// Mitsubishi GX Works2 project: 3. teaching   PLC: Q03UDV

PROGRAM MAIN
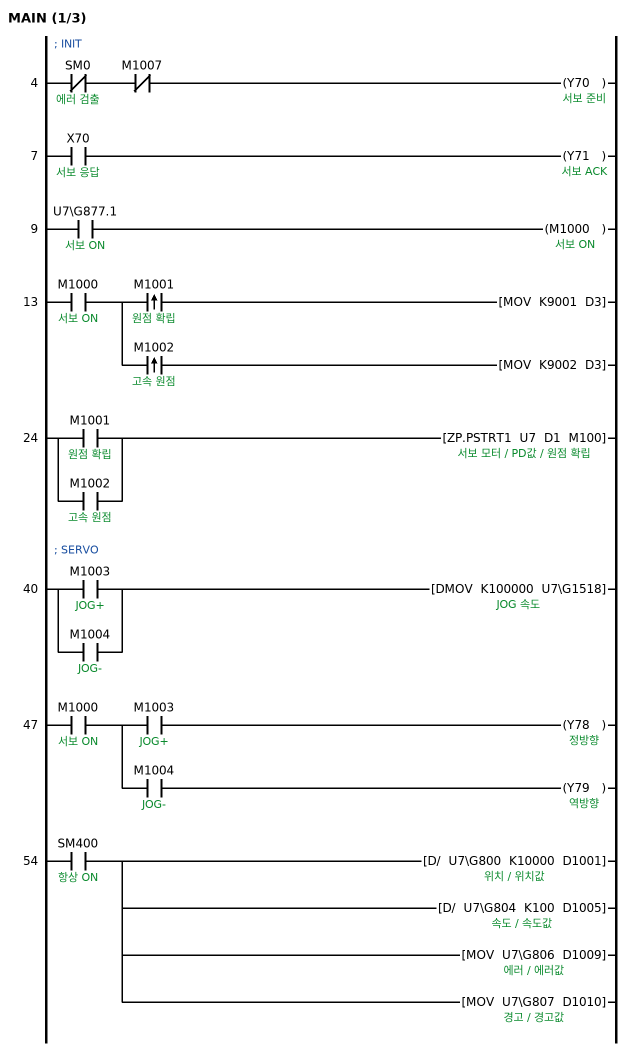
; INIT
4     LDI     SM0  ; 에러 검출
      ANI     M1007
      OUT     Y70  ; 서보 준비
7     LD      X70  ; 서보 응답
      OUT     Y71  ; 서보 ACK
9     LD      U7\G877.1  ; 서보 ON
      OUT     M1000  ; 서보 ON
13    LD      M1000  ; 서보 ON
      MPS
      ANDP    M1001  ; 원점 확립
      MOV     K9001 D3
      MPP
      ANDP    M1002  ; 고속 원점
      MOV     K9002 D3
24    LD      M1001  ; 원점 확립
      OR      M1002  ; 고속 원점
      ZP.PSTRT1 U7 D1 M100  ; 서보 모터 / PD값 / 원점 확립
; SERVO
40    LD      M1003  ; JOG+
      OR      M1004  ; JOG-
      DMOV    K100000 U7\G1518  ; JOG 속도
47    LD      M1000  ; 서보 ON
      MPS
      AND     M1003  ; JOG+
      OUT     Y78  ; 정방향
      MPP
      AND     M1004  ; JOG-
      OUT     Y79  ; 역방향
54    LD      SM400  ; 항상 ON
      D/      U7\G800 K10000 D1001  ; 위치 / 위치값
      D/      U7\G804 K100 D1005  ; 속도 / 속도값
      MOV     U7\G806 D1009  ; 에러 / 에러값
      MOV     U7\G807 D1010  ; 경고 / 경고값
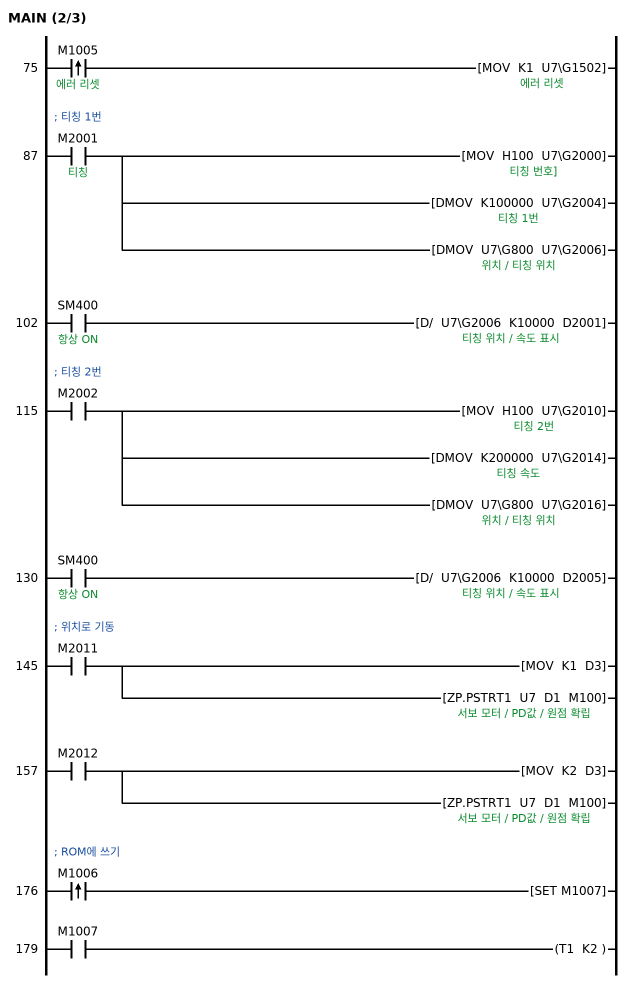
75    LDP     M1005  ; 에러 리셋
      MOV     K1 U7\G1502  ; 에러 리셋
; 티칭 1번
87    LD      M2001  ; 티칭
      MOV     H100 U7\G2000  ; 티칭 번호]
      DMOV    K100000 U7\G2004  ; 티칭 1번
      DMOV    U7\G800 U7\G2006  ; 티칭 위치
102   LD      SM400  ; 항상 ON
      D/      U7\G2006 K10000 D2001  ; 속도 표시
; 티칭 2번
115   LD      M2002
      MOV     H100 U7\G2010  ; 티칭 2번
      DMOV    K200000 U7\G2014  ; 티칭 속도
      DMOV    U7\G800 U7\G2016  ; 티칭 위치
130   LD      SM400  ; 항상 ON
      D/      U7\G2006 K10000 D2005  ; 속도 표시
; 위치로 기동
145   LD      M2011
      MOV     K1 D3
      ZP.PSTRT1 U7 D1 M100
157   LD      M2012
      MOV     K2 D3
      ZP.PSTRT1 U7 D1 M100
; ROM에 쓰기
176   LDP     M1006
      SET     M1007
179   LD      M1007
      OUT     T1 K2
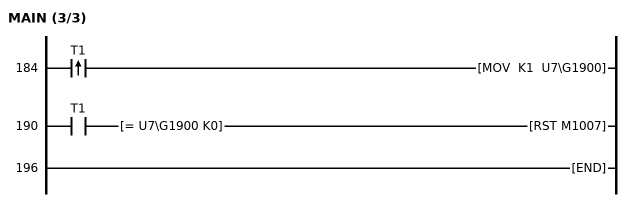
184   LDP     T1
      MOV     K1 U7\G1900
190   LD      T1
      AND=    U7\G1900 K0
      RST     M1007
196   END
END_PROGRAM

// device comments not shown above
X0  ; 공급 후진
X1  ; 공급 전진
X2  ; 분배 후진
X3  ; 분배 전진
X4  ; 가공 상승
X15  ; PB1
X16  ; PB2
X17  ; PB3
X1C  ; Toggle
Y20  ; 공급+
Y21  ; 공급-
Y22  ; 분배+
Y23  ; 분배-
M1  ; 공급+
M2  ; 공급-
M3  ; 분배+
M4  ; 분배-
M10  ; 무한 반복
P1  ; STOP
